(* IEC 61131-3 sources: Industry-PLC-LLM/data/PLCBEAD_repo/PLCBEAD_PLCEmbed-main/PLC-BEAD/Source/GEB/_ARRAY_MUL, 1 file *)

(* ---- _ARRAY_MUL.ST ---- *)
TYPE
	oscat_PT_ARRAY: ARRAY [1..100] OF REAL;
END_TYPE

FUNCTION_BLOCK ARRAY_MUL2
	VAR_IN_OUT
		PT :	oscat_PT_ARRAY;
	END_VAR
	VAR_INPUT
		SIZE :	UINT;
		X :	REAL;
	END_VAR
	VAR_OUTPUT
		ARRAY_MUL :	BOOL;
	END_VAR
	VAR
		i :	INT;
		STOP :	INT;
	END_VAR

	STOP :=LIMIT_INT(1,UINT_TO_INT(SIZE),1000);
	FOR i := 1 TO STOP DO
		PT[i] := PT[i] * X;
	END_FOR;
	ARRAY_MUL := TRUE;

END_FUNCTION_BLOCK

PROGRAM program0
  VAR
    LocalVar0 : oscat_PT_ARRAY;
    LocalVaR1  : UINT;
	LocalVaR2 : REAL;
	LocalOUT  : BOOL;
	func_block : ARRAY_MUL2;
  END_VAR
	func_block(PT := LocalVar0, SIZE := LocalVaR1 , X:= LocalVaR2);
	LocalOUT := func_block.ARRAY_MUL;
END_PROGRAM
